(* IEC 61131-3 sources: Industry-PLC-LLM/data/PLCBEAD_repo/PLCBEAD_PLCEmbed-main/PLC-BEAD/Source/GEB/Network_TN_SC_AREA_RESTORE, 1 file *)

(* ---- TN_SC_AREA_RESTORE.ST ---- *)
TYPE
  bya_TN_CHAR:       	ARRAY [0..1919] OF BYTE;
  bya_TN_BACKUP:     	ARRAY [0..1919] OF BYTE;
  bya_TN_COLOR:      	ARRAY [0..1919] OF BYTE;
  bya_TN_Line_Update:	ARRAY [0..23]   OF BOOL;

  us_TN_SCREEN :
  STRUCT
		bya_CHAR:			bya_TN_CHAR;
		bya_COLOR:			bya_TN_COLOR;
		bya_BACKUP:			bya_TN_BACKUP;
		bya_Line_Update:	bya_TN_Line_Update;

		by_Input_Exten_Code:    BYTE;
		by_Input_ASCII_Code:    BYTE;
		bo_Input_ASCII_IsNum:   BOOL;
		in_Page_Number:        	INT;                (* aktive Seiten-Nr.              *)
		in_Cursor_X:           	INT;                (* Cursor X-POSition              *)
		in_Cursor_Y:           	INT;                (* Cursor Y-POSition              *)
		in_EOS_Offset:         	INT;                (* End of String Offset           *)
		by_Clear_Screen_Attr:  	BYTE;               (* Clear-Screen Attr              *)
		bo_Clear_Screen:       	BOOL;               (* Clear-Screen ausl�sen          *)
		bo_Modal_Dialog:       	BOOL;               (* Modaler Dialog ist aktiv       *)
		bo_Menue_Bar_Dialog:   	BOOL;               (* Menue Dialog ist aktiv         *)

  END_STRUCT;
END_TYPE

FUNCTION TN_SC_XY2_ERROR:BOOL

	VAR_INPUT
		X1 :	INT;
		Y1 :	INT;
		X2 :	INT;
		Y2 :	INT;
	END_VAR

	TN_SC_XY2_ERROR := Y1 < 0 OR X1 < 0 OR Y2 < 0 OR X2 < 0 OR Y1 > 23 OR X1 > 79 OR Y2 > 23 OR X2 > 79;

END_FUNCTION

FUNCTION _BYTE_TO_INT:INT
	VAR_INPUT
		IN :	BYTE;
	END_VAR

	_BYTE_TO_INT := USINT_TO_INT(BYTE_TO_USINT(IN));
END_FUNCTION

FUNCTION_BLOCK TN_SC_AREA_RESTORE_Block

  VAR
    in_Offset_1 :	INT;
    in_Offset_2 :	INT;
    in_Y :	INT;
    in_X :	INT;
    in_Y1 :	INT;
    in_X1 :	INT;
    in_Y2 :	INT;
    in_X2 :	INT;
  END_VAR

  VAR_IN_OUT
    Xus_TN_SCREEN :	us_TN_SCREEN;
  END_VAR

  IF Xus_TN_SCREEN.bya_BACKUP[0] > BYTE#00 THEN

    in_X1 := _BYTE_TO_INT(Xus_TN_SCREEN.bya_BACKUP[1]);
    in_Y1 := _BYTE_TO_INT(Xus_TN_SCREEN.bya_BACKUP[2]);
    in_X2 := _BYTE_TO_INT(Xus_TN_SCREEN.bya_BACKUP[3]);
    in_Y2 := _BYTE_TO_INT(Xus_TN_SCREEN.bya_BACKUP[4]);

    IF TN_SC_XY2_ERROR(in_X1,in_Y1,in_X2,in_Y2) THEN RETURN; END_IF;
    in_Offset_2 := 5;

    FOR in_Y := in_Y1 TO in_Y2 DO

      Xus_TN_SCREEN.bya_Line_Update[in_Y] := TRUE;
      in_Offset_1 := (in_Y * 80) + in_X1;

      FOR in_X := in_X1 TO in_X2 DO

        Xus_TN_SCREEN.bya_CHAR[in_Offset_1] := Xus_TN_SCREEN.bya_BACKUP[in_Offset_2];
        in_Offset_2 := in_Offset_2 + INT#01;

        Xus_TN_SCREEN.bya_COLOR[in_Offset_1] := Xus_TN_SCREEN.bya_BACKUP[in_Offset_2];
        in_Offset_2 := in_Offset_2 + INT#01;
        in_Offset_1 := in_Offset_1 + INT#01;

      END_FOR;

    END_FOR;

    Xus_TN_SCREEN.bya_BACKUP[0] := BYTE#00;
  END_IF;

END_FUNCTION_BLOCK

PROGRAM program0
	VAR
		Xus_TN_SCREEN :	us_TN_SCREEN;

		func_block : TN_SC_AREA_RESTORE_Block;
	END_VAR
	func_block.Xus_TN_SCREEN := Xus_TN_SCREEN;

	func_block();
	Xus_TN_SCREEN  := func_block.Xus_TN_SCREEN;
END_PROGRAM
